PROGRAM MAIN
VAR
END_VAR

//----------------------------------------程序调用----------------------------------------------
InputLink();
S01_Loading();
S02_LidInjecting();
S03_LidChecking();
S04_AluCovering();
S05_Adjusting();
S06_Cutting();
S07_BoxCarrying();
S08_MainLine();
S09_CardCarrying();
S10_BeltCarrying();
S11_Packing();
S12_PreLine();
S13_Labeling();
S14_LabelChecking();
S15_NG();
S16_Unloading();

ControlMachine();
CallStandard();
CommWithPC();
OutputLink();
LightsTest();

END_PROGRAM

(* stored: Version 1.1.0.1, ProductVersion 3.1.4024.9
   POU MAIN: Id {e1b95b3d-d72e-4236-b2e9-ad4cda4ca0ec}, SpecialFunc None *)
